FUNCTION_BLOCK FB_PalletizerElevator EXTENDS FB_Elevator
VAR_INPUT
END_VAR
VAR_OUTPUT
	isMoving : BOOL;
END_VAR
VAR
	fbElevatorMoving : FB_Sensor;
	
END_VAR

isMoving := fbElevatorMoving.bSignal;

METHOD MoveDown : BOOL
VAR_INPUT
END_VAR
END_METHOD

METHOD MoveUp : BOOL
VAR_INPUT
END_VAR
END_METHOD

METHOD StepDown : BOOL
VAR_INPUT
END_VAR
END_METHOD

METHOD StepUp : BOOL
VAR_INPUT
END_VAR
END_METHOD

END_FUNCTION_BLOCK

(* stored: Version 1.1.0.1, ProductVersion 3.1.4024.0
   POU FB_PalletizerElevator: Id {bd2ea0f4-c169-461a-88aa-19be27edaaa5}, SpecialFunc None
   Method MoveDown: Id {73b801bf-e72e-41ab-ac7b-579ada3843c5}
   Method MoveUp: Id {c7f781fc-6698-47a1-8530-f8c7485ab296}
   Method StepDown: Id {3890aa0b-5570-4bd0-b4f2-65dbeb3ba42b}
   Method StepUp: Id {3875e7be-0bef-425d-a77a-139b2a0aa8ce} *)
